PROGRAM STPOU
VAR
	// Start Button
	btnStart: BOOL;
	// Stop Button
	btnStop: BOOL;
	// Motor Starter Coil
	Coil: BOOL;
END_VAR

Coil := NOT btnStop AND (btnStart OR Coil);

END_PROGRAM

(* stored: Version 1.1.0.1, ProductVersion 3.1.4024.15
   POU STPOU: Id {efb8ad37-cf68-421c-8534-f1f910a9749d}, SpecialFunc None *)
